PROGRAM Test
VAR
END_VAR

END_PROGRAM

(* stored: Version 1.1.0.1
   POU Test: Id {1debf982-2c16-434e-985d-59b47fe99478}, SpecialFunc None *)
